// TIA Portal V20 export
// export: Created 2026-07-10T11:12:01.1919651Z, ExportSetting WithDefaults, DisplayName Totally Integrated Automation Portal, DisplayVersion V20, DisplayName TIA Portal Openness, DisplayVersion V20, DisplayName TIA Portal Version Control Interface, DisplayVersion V20, DisplayName STEP 7 Professional, DisplayVersion V20, DisplayName STEP 7 Safety, DisplayVersion V20, DisplayName WinCC Basic/Comfort/Advanced, DisplayVersion V20, DisplayName WinCC Unified, DisplayVersion V20
ORGANIZATION_BLOCK "Main"   // OB1, SCL, ProgramCycle
TITLE = "Main Program Sweep (Cycle)"
{ S7_Optimized_Access := 'TRUE' }
VERSION : 0.1
// stored: AutoNumber true, IsIECCheckEnabled false, SetENOAutomatically false
   VAR_INPUT
      Initial_Call : Bool;   // Initial call of this OB
      Remanence : Bool;   // =True, if remanent data are available
   END_VAR
BEGIN
   "SystemClock"();
   "Inputs_DB"();
   "WaterCounter_DB"();
   "HMI_DB"();
   "Alarms_DB"();
   "WorkModeCycle_DB"();
   "Dampers_DB"();
   "Weighting_DB"();
   "MBServer_DB"();
   "ModbusClO2_DB"();
   "ChlorMode_DB"();

   "MB".Table.Chlor_Setpoint := "MB".Table.ChlorationParams.ActualDose;
   "MB".Table.Chlor_PulseWeight := "MB".Table.MeasuredChlor;
END_ORGANIZATION_BLOCK
